FUNCTION_BLOCK BASIC_SEND_ENQ (* Basic Function Block Type *)
  (* Standard: 61499-2 *)
  (* Version 0.0, 2015-11-04, 4DIAC-IDE, 4DIAC-Consortium *)
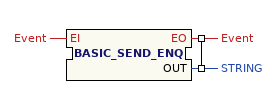
  EVENT_INPUT
    EI;
  END_EVENT
  EVENT_OUTPUT
    EO WITH OUT;
  END_EVENT
  VAR_OUTPUT
    OUT : STRING;
  END_VAR
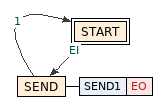
  EC_STATES
    START; (* Initial State *)
    SEND : SEND1 -> EO; (* Normal execution *)
  END_STATES
  EC_TRANSITIONS
    START TO SEND := EI;
    SEND TO START := 1;
  END_TRANSITIONS
  ALGORITHM SEND1 IN ST: (* Normally executed algorithm *)
OUT:='\x05';
  END_ALGORITHM
END_FUNCTION_BLOCK
